Fanuc TP program (LS listing): MOTION.LS

/PROG  MOTION
/ATTR
OWNER		= MNEDITOR;
COMMENT		= "";
PROG_SIZE	= 182;
CREATE		= DATE 17-10-19  TIME 13:19:58;
MODIFIED	= DATE 17-10-19  TIME 13:21:10;
FILE_NAME	= ;
VERSION		= 0;
LINE_COUNT	= 4;
MEMORY_SIZE	= 546;
PROTECT		= READ_WRITE;
TCD:  STACK_SIZE	= 0,
      TASK_PRIORITY	= 50,
      TIME_SLICE	= 0,
      BUSY_LAMP_OFF	= 0,
      ABORT_REQUEST	= 0,
      PAUSE_REQUEST	= 0;
DEFAULT_GROUP	= 1,*,*,*,*;
CONTROL_CODE	= 00000000 00000000;
/MN
   1:  PAYLOAD[1] ;
   2:   ;
   3:   ;
   4:  CALL GET_HOME    ;
/POS
/END
